{attribute 'qualified_only'}
{attribute 'strict'}
TYPE E_Joystick :
(
	JoyX,
	JoyY
);
END_TYPE

(* stored: Version 1.1.0.1, ProductVersion 3.1.4024.9
   DUT E_Joystick: Id {376804ef-6514-4794-bc9c-72fa8cecea07} *)
